{attribute 'qualified_only'}
{attribute 'strict'}
TYPE E_Hmi_ButtonBehaviour :
(
	MomentaryOn := 0,
	MomentaryOff := 1,
	Toggle := 2,
	Set := 3,
	Reset := 4
)UINT;
END_TYPE

(* stored: Version 1.1.0.1, ProductVersion 3.1.4024.10
   DUT E_Hmi_ButtonBehaviour: Id {28bc2804-25f9-43db-84f8-da9946bdddf2} *)
